(* IEC 61131-3 sources: moqui-plc/simatic-ax/src/moqui/runtime/component/mantle-hvac/src/main/mantle/hvac, 4 files *)

(* ---- MainStatus.st ---- *)
TYPE MainStatus : (
	Standby,
    Ventilation,
    Cooling,
    Heating,
	Drying,
    Fault
); END_TYPE

(* ---- Main.st ---- *)
(*
 * NOTE: In general, the Main component implements the control logic of automated industrial systems (Finite State Machine - FSM)
 * using hierarchical control architectures. It separates control policies from implementation mechanisms,
 * and diagnostic mechanisms from failure/error reaction and system reset policies.
*)

(* Example of a supervisor FSM for a civil HVAC air-handling unit (AHU).
 *
 * Topology:
 *   Mode A Thermostat cooling -> Cooling
 *   Mode B Cooling with RH% dehumidification -> Cooling  (rhControlEnabled=TRUE)
 *   Mode C Winter heating -> Heating
 *   Mode D Heating with RH% control -> Heating (rhControlEnabled=TRUE)
 *   Mode E Interval dehumidification (on/off) -> Drying
 *   Mode F Dehumidification by RH% target -> Drying (rhControlEnabled=TRUE)
 *
 * Output function - which device groups are enabled per state:
 *
 *   State          Cold Group   Hot Group   AHU Fan   Air Flow
 *   -
 *   Standby            OFF         OFF        OFF       OFF
 *   Ventilation        OFF         OFF        ON        ON
 *   Cooling            ON          OFF        ON        ON
 *   Heating            OFF         ON         ON        ON
 *   Drying             ON          ON         ON        ON
 *   Fault              OFF         OFF        OFF       OFF
 *
 * MainRuleEngine generates transition requests; Main consumes them.
 * DeviceManager orchestrates the individual device FBs.
 *
 * Call order in the PLC task:
 *   InputSignalUpdate -> Main -> DeviceManager -> OutputSignalUpdate
 *)
FUNCTION_BLOCK Main
	VAR_EXTERNAL
		clks : Clocks;
		dev : DeviceFacade;
	END_VAR
	VAR_INPUT
		operationType : OperatingMode;
		enable : BOOL;
		deviceConfigContextResetRequest : BOOL := FALSE;
	END_VAR
	VAR_OUTPUT
		done : BOOL;
		error : BOOL;
	END_VAR
	VAR CONSTANT
		componentName : STRING := 'hvac';
	END_VAR
	VAR
		(* Logger facade *)
		logger : LoggerFacade;
		(* FSM transition logic *)
		ruleEngine : MainRuleEngine;
		(* Define a nested FSMs for managing air distribution subsystem. *)
		airDistribCtrl : AirDistributionController;
		(* HAL manager *)
		deviceManager : DeviceManager;
	END_VAR

	(* Logger facade init *)
	logger.enable := TRUE; logger.loggerName := componentName;

	IF NOT enable THEN RETURN; END_IF;

	(* Init: device setup and configuration *)
	IF (operationType = OperatingMode#Init) THEN
		logger(message := 'Setup and configuration of all devices.', level := LogLevel#DEBUG);
		(*
	     * The static device configuration parameters are mapped directly by the device config manager (recipe manager),
		 * while only the dynamic parameters are mapped below in the standby status.
		 *)
		(* Reset signal manager *)
		dev.signalMgmt(operationType := SignalMgmtOperatingMode#Reset, loggerName := componentName);
		dev.status := MainStatus#Standby;
		dev.actualRuntime := UDINT#0;
		dev.actualBreakDuration := UDINT#0;
		dev.processActualDuration := UDINT#0;
		dev.processRemainingDuration := UDINT#0;
		dev.timeBreakEnabled := FALSE;
		dev.isCompleted := FALSE;
		airDistribCtrl(operationType := OperatingMode#Init, enable := FALSE, clock1s := FALSE);
		done := FALSE;
	ELSIF deviceConfigContextResetRequest THEN
		logger(message := 'Reset HVAC device config context.', level := LogLevel#DEBUG);
		(*
	     * Lightweight reset between recipes: keep device init/homing in the Init path,
		 * but clear runtime state inherited from the previous device config.
	     *)
		dev.status := MainStatus#Standby;
		dev.lastStatus := MainStatus#Standby;
		dev.actualRuntime := UDINT#0;
		dev.actualBreakDuration := UDINT#0;
		dev.processActualDuration := UDINT#0;
		dev.processRemainingDuration := UDINT#0;
		dev.timeBreakEnabled := FALSE;
		dev.isCompleted := FALSE;
		airDistribCtrl(operationType := OperatingMode#Init, enable := FALSE, clock1s := FALSE);
		done := FALSE;
	ELSE
		(* FSM transition-condition rule engine *)
		logger(message := 'Run FSM transition-condition logic.', level := LogLevel#DEBUG);
		ruleEngine(operationType := operationType);
	END_IF;

		(*
		 * Preserve the originating phase while idling in Standby so thermostat-driven
		 * Heating/Cooling recipes can stop/start repeatedly until isCompleted becomes TRUE.
		 * Init still stamps Standby, which keeps fresh-start logic for a newly loaded recipe.
	     *)
		IF (operationType = OperatingMode#Init) OR (dev.status <> MainStatus#Standby) THEN
			dev.lastStatus := dev.status;
		END_IF;

	(* Fault overrides any other state *)
	IF dev.faultRequest THEN dev.status := MainStatus#Fault; END_IF;

	(* Main FSM - Output function + State-update function *)
	logger(message := 'Run Main FSM.', level := LogLevel#DEBUG);
	CASE dev.status OF
	    (* Standby / Homing: all groups off, wait for the next phase request. *)
		MainStatus#Standby :
			logger(message := 'Standby.', level := LogLevel#DEBUG);
			dev.standbyRequest := FALSE;

			(* FSM Output function - everything disabled *)
			dev.coldGroupEnableRequest := FALSE;
			dev.coldGroupDisableRequest := TRUE;
			dev.hotGroupEnableRequest := FALSE;
			dev.hotGroupDisableRequest := TRUE;
			dev.ahuFanEnableRequest := FALSE;
			dev.airFlowEnableRequest := FALSE;
			dev.airFlowDisableRequest := TRUE;

			(* FSM status update function *)
			IF dev.ventilationRequest THEN
				dev.status := MainStatus#Ventilation;
			ELSIF dev.coolingRequest THEN
				dev.status := MainStatus#Cooling;
			ELSIF dev.heatingRequest THEN
				dev.status := MainStatus#Heating;
			ELSIF dev.dryingRequest THEN
				dev.status := MainStatus#Drying;
			END_IF;

	    (* Ventilation: AHU + air flow control only - no temperature conditioning. *)
		MainStatus#Ventilation :
			logger(message := 'Ventilation.', level := LogLevel#DEBUG);
			dev.ventilationRequest := FALSE;

			(* FSM output function *)
			dev.coldGroupEnableRequest := FALSE;
			dev.coldGroupDisableRequest := TRUE;
			dev.hotGroupEnableRequest := FALSE;
			dev.hotGroupDisableRequest := TRUE;
			dev.ahuFanEnableRequest := TRUE;
			dev.airFlowEnableRequest := TRUE;
			dev.airFlowDisableRequest := FALSE;

			(* FSM status update function *)
			IF dev.standbyRequest THEN
				dev.status := MainStatus#Standby;
			ELSIF dev.coolingRequest THEN
				dev.status := MainStatus#Cooling;
			ELSIF dev.heatingRequest THEN
				dev.status := MainStatus#Heating;
			ELSIF dev.dryingRequest THEN
				dev.status := MainStatus#Drying;
			END_IF;

	    (*
	     * Cooling: cold group + AHU + air flow control.
	     * Phase 0 (no RH ctrl) and Phase 1 (with RH ctrl, rhControlEnabled=TRUE).
	     * In Phase 1 the hot group is also enabled to post-heat after dehumidification;
	     * that secondary enable is issued by MainRuleEngine via heatingRequest/dryingRequest
	     * transitions rather than here, keeping output function clean.
	     *)
		MainStatus#Cooling :
			logger(message := 'Cooling.', level := LogLevel#DEBUG);
			dev.coolingRequest := FALSE;

			(* FSM output function *)
			dev.coldGroupEnableRequest := TRUE;
			dev.coldGroupDisableRequest := FALSE;
			dev.hotGroupEnableRequest := FALSE;
			dev.hotGroupDisableRequest := TRUE;
			dev.ahuFanEnableRequest := TRUE;
			dev.airFlowEnableRequest := TRUE;
			dev.airFlowDisableRequest := FALSE;

			(* FSM status update function *)
			IF dev.standbyRequest THEN
				dev.status := MainStatus#Standby;
			ELSIF dev.dryingRequest THEN
				dev.status := MainStatus#Drying;
			ELSIF dev.ventilationRequest THEN
				dev.status := MainStatus#Ventilation;
			END_IF;

	    (*
	     * Heating: hot group + AHU + air flow control.
	     * Phase 2 (no RH ctrl) and Phase 3 (with RH ctrl).
	     *)
		MainStatus#Heating :
			logger(message := 'Heating.', level := LogLevel#DEBUG);
			dev.heatingRequest := FALSE;

			(* FSM output function *)
			dev.coldGroupEnableRequest := FALSE;
			dev.coldGroupDisableRequest := TRUE;
			dev.hotGroupEnableRequest := TRUE;
			dev.hotGroupDisableRequest := FALSE;
			dev.ahuFanEnableRequest := TRUE;
			dev.airFlowEnableRequest := TRUE;
			dev.airFlowDisableRequest := FALSE;

			(* FSM status update function *)
			IF dev.standbyRequest THEN
				dev.status := MainStatus#Standby;
			ELSIF dev.dryingRequest THEN
				dev.status := MainStatus#Drying;
			ELSIF dev.ventilationRequest THEN
				dev.status := MainStatus#Ventilation;
			END_IF;

	    (*
	     * Drying: cold + hot + AHU + air flow control.
	     * Phase 4 (time-based run/break) and Phase 5 (RH% controlled).
	     * During break the rule engine transitions to Standby; returns here
	     * when the break is complete.
	     *)
		MainStatus#Drying :
			logger(message := 'Drying.', level := LogLevel#DEBUG);
			dev.dryingRequest := FALSE;

			(* FSM output function *)
			dev.coldGroupEnableRequest := TRUE;
			dev.coldGroupDisableRequest := FALSE;
			dev.hotGroupEnableRequest := TRUE;
			dev.hotGroupDisableRequest := FALSE;
			dev.ahuFanEnableRequest := TRUE;
			dev.airFlowEnableRequest := TRUE;
			dev.airFlowDisableRequest := FALSE;

			(* FSM status update function *)
			IF dev.standbyRequest THEN
				dev.status := MainStatus#Standby;
			ELSIF dev.heatingRequest THEN
				dev.status := MainStatus#Heating;
			ELSIF dev.coolingRequest THEN
				dev.status := MainStatus#Cooling;
			ELSIF dev.ventilationRequest THEN
				dev.status := MainStatus#Ventilation;
			END_IF;

	    (* Fault: all groups off; wait for signal manager to clear all alarms. *)
		MainStatus#Fault :
			logger(message := 'Fault.', level := LogLevel#DEBUG);
			dev.faultRequest := FALSE;

			(* FSM output function *)
			error := TRUE;
			dev.coldGroupEnableRequest := FALSE;
			dev.coldGroupDisableRequest := TRUE;
			dev.hotGroupEnableRequest := FALSE;
			dev.hotGroupDisableRequest := TRUE;
			dev.ahuFanEnableRequest := FALSE;
			dev.airFlowEnableRequest := FALSE;
			dev.airFlowDisableRequest := TRUE;

			(* Return to Standby only when all alarms have been cleared *)
			IF (dev.signalMgmt.cumulativeOutputAction = DWORD#16#0000) THEN
				error := FALSE;
				dev.status := MainStatus#Standby;
			END_IF;
	END_CASE;

	(*
	 * Air distribution is a subordinate subsystem:
	 * it runs only when the main FSM requests air flow and the recipe explicitly
	 * enables alternating high/low air distribution.
	 *)
	airDistribCtrl(
		operationType := operationType,
		enable := dev.airFlowEnableRequest AND dev.airDistributionEnabled,
		clock1s := clks.clock1s);

	done := dev.isCompleted;

	(* Device orchestration (HAL) *)
	logger(message := 'Update HVAC devices.', level := LogLevel#DEBUG);
	deviceManager(operationType := operationType);
	END_FUNCTION_BLOCK

(* ---- MainRuleEngine.st ---- *)
(*
 * MainRuleEngine - transition-condition logic for the HVAC supervisor FSM.
 *
 * Responsibilities:
 *   1. Reset transition requests to safe defaults.
 *   2. Run the signal management engine (fault / alarm / warning detection).
 *   3. Compute boolean predicates from sensor feedback and recipe setpoints.
 *   4. Implement the per-state transition-condition rules.
 *
 * Default / persistence convention
 * At the top of every scan standbyRequest is set TRUE (safe default).
 * Each ACTIVE-state CASE block MUST:
 *   • Set standbyRequest := FALSE (keep current state) in the ELSE branch.
 *   • Set standbyRequest := TRUE (or leave as-is) when an EXIT condition is met.
 *   • Set standbyRequest := FALSE and another*Request := TRUE to switch phase.
 *
 * Without the ELSE branch the system would exit any active state to Standby
 * on the very first scan - a single-scan flash rather than a persistent phase.
 *
 * Process phases:
 *   Phase 0 Thermostat Cooling -> Cooling
 *   Phase 1 Cooling with RH% control -> Cooling (rhControlEnabled)
 *   Phase 2 Heating without RH% control -> Heating
 *   Phase 3 Heating with RH% control -> Heating (rhControlEnabled)
 *   Phase 4 Timed Drying (on/off) -> Drying <-> Standby (break)
 *   Phase 5 Drying with RH% control -> Drying (rhControlEnabled)
 *
 * Duct safety (duct sensors):
 *   The duct T+RH sensor monitors supply-air conditions before the air
 *   enters the curing room. Limit violations raise alarms to protect
 *   product (≈ €80-90 k of salami/prosciutto on trolleys).
 *   ductTempOverMax -> air too hot -> ImmediateStop (protects product)
 *   ductTempUnderMin -> air too cold -> ImmediateStop (protects product)
 *   ductRhOverMax -> saturated -> Warning only (condensation risk)
 *)
FUNCTION_BLOCK MainRuleEngine
	VAR_EXTERNAL
		clks : Clocks;
		dev : DeviceFacade;
	END_VAR
	VAR_INPUT
		operationType : OperatingMode := OperatingMode#Run;
	END_VAR
	VAR_OUTPUT
		error : BOOL;
	END_VAR
	VAR
		(* Device diagnostics *)
		deviceDiags : DeviceDiagnostics;
		tempDeviation : REAL;
		rhDeviation : REAL;
	END_VAR

	(* Reset transition requests to safe defaults.
	 *
	 * standbyRequest = TRUE  -> return to / stay in Standby (safe default).
	 * Active-state CASE blocks override to FALSE to keep the current phase alive,
	 * or set another *Request to switch phases.
	 *)
	dev.faultRequest := FALSE;
	dev.standbyRequest := TRUE;
	dev.heatingRequest := FALSE;
	dev.coolingRequest := FALSE;
	dev.ventilationRequest := FALSE;
	dev.dryingRequest := FALSE;

	deviceDiags(operationType := operationType, error => error);

	(* Compute sensor predicates *)

	(* Process temperature sensor *)
	dev.tempInRange := (dev.tempFeedback >= dev.tempMin + dev.tempHysteresis)
		AND (dev.tempFeedback <= dev.tempMax - dev.tempHysteresis);
	tempDeviation := dev.tempFeedback - dev.tempSetpoint;
	IF tempDeviation < REAL#0.0 THEN
		tempDeviation := -tempDeviation;
	END_IF;
	dev.tempAtSetpoint := tempDeviation <= dev.tempHysteresis;
	dev.tempOverMax := dev.tempFeedback > dev.tempMax;
	dev.tempOverMin := dev.tempFeedback > dev.tempMin;
	dev.tempUnderMin := dev.tempFeedback < dev.tempMin;
	dev.tempUnderMax := dev.tempFeedback < dev.tempMax;
	(* Process RH sensor *)
	rhDeviation := dev.rhFeedback - dev.rhSetpoint;
	IF rhDeviation < REAL#0.0 THEN
		rhDeviation := -rhDeviation;
	END_IF;
	dev.rhAtSetpoint := rhDeviation <= dev.rhHysteresis;
	dev.rhOverMax := dev.rhFeedback > dev.rhMax - dev.rhHysteresis;
	dev.rhUnderMin := dev.rhFeedback < dev.rhMin + dev.rhHysteresis;
	dev.rhOverMin := dev.rhFeedback > dev.rhMin;
	dev.rhUnderMax := dev.rhFeedback < dev.rhMax;

	(* Duct sensor - safety predicates *)
	dev.ductTempOverMax := dev.ductTempFeedback > dev.ductTempMax;
	dev.ductTempUnderMin := dev.ductTempFeedback < dev.ductTempMin;
	dev.ductRhOverMax := dev.ductRhFeedback > dev.ductRhMax;

	(*
	 * Process timing - run / break cycle.
	 *
	 * processActualDuration must NOT advance while the FSM is in Standby
	 * waiting for a phase to start (i.e. not in a break).
	 * If it did, isCompleted could fire while the process has not yet begun,
	 * causing the phase to complete immediately without doing any work.
	 *
	 * Counting rules:
	 *   Break  (timeBreakEnabled=TRUE, status=Standby): advance processActualDuration + actualBreakDuration.
	 *   Active (status ≠ Standby):                      advance processActualDuration + actualRuntime.
	 *   Idle   (status=Standby, NOT timeBreakEnabled):  no counters advance.
	 *)
	IF clks.clock1s THEN
		IF dev.timeBreakEnabled AND dev.status = MainStatus#Standby THEN
			(* Break counting *)
			dev.processActualDuration := dev.processActualDuration + UDINT#1;
			dev.actualBreakDuration := dev.actualBreakDuration + UDINT#1;
			IF dev.estimatedBreakDuration > UDINT#0 THEN
				(* Break ends when both minimum and estimated durations are met; reset counters for next run *)
				IF (dev.actualBreakDuration >= dev.estimatedBreakDuration)
						AND (dev.actualBreakDuration >= dev.minBreakDuration) THEN
					dev.timeBreakEnabled := FALSE;
					dev.actualRuntime := UDINT#0;
					dev.actualBreakDuration := UDINT#0;
				END_IF;
			END_IF;
		ELSIF dev.status <> MainStatus#Standby THEN
			(* Active run counting - only while the FSM is in an active phase state *)
			dev.processActualDuration := dev.processActualDuration + UDINT#1;
			dev.actualRuntime := dev.actualRuntime + UDINT#1;
			IF dev.estimatedRuntime > UDINT#0 THEN
				dev.processRemainingDuration := dev.processEstimatedDuration - dev.processActualDuration;
				IF NOT dev.timeBreakEnabled
						AND (dev.actualRuntime >= dev.estimatedRuntime)
						AND (dev.actualRuntime >= dev.minRuntime) THEN
					dev.timeBreakEnabled := TRUE;
					dev.actualBreakDuration := UDINT#0;
				END_IF;
			END_IF;
		ELSIF (dev.lastStatus = MainStatus#Cooling OR dev.lastStatus = MainStatus#Heating)
				AND NOT dev.isCompleted THEN
			(* Thermostat dwell between active cycles counts toward phase duration,
			 * but does not count as active runtime. *)
			dev.processActualDuration := dev.processActualDuration + UDINT#1;
			IF dev.processEstimatedDuration > UDINT#0 THEN
				dev.processRemainingDuration := dev.processEstimatedDuration - dev.processActualDuration;
			END_IF;
		END_IF;

		(* isCompleted is independent of the run/break cycle:
		 * a phase with only processEstimatedDuration set (no run/break) must also complete. *)
		IF dev.processEstimatedDuration > UDINT#0 THEN
			dev.isCompleted :=
				(dev.processActualDuration >= dev.processEstimatedDuration)
				AND (dev.processActualDuration >= dev.processMinDuration);
		END_IF;
	END_IF;

	(* Fault gate *)
	IF error OR ((dev.signalMgmt.cumulativeOutputAction AND DWORD#16#0002) <> DWORD#16#0000) THEN
		dev.faultRequest := TRUE;
		RETURN;
	END_IF;

	(*
	 * Transition-condition rule engine
	 *
	 * Persistence rule: every active-state CASE MUST end with
	 *   ELSE dev.standbyRequest := FALSE; [ keep current state alive ]
	 * to prevent the scan-level default (standbyRequest=TRUE) from immediately
	 * bouncing the FSM back to Standby before the exit condition is reached.
	 *)
	CASE dev.status OF
	    (*
	     * Standby - decide next phase.
	     * Default standbyRequest=TRUE keeps the system here.
	     * Override when an external condition requires re-entering a phase.
	     *)
		MainStatus#Standby :
			(*
			 * Transition-condition evaluation order:
			 *   1. Safety overrides (cooling/heating if temperature out of limits).
			 *   2. Phase-resume conditions (drying after break, thawing).
			 *   3. Fresh-start drying (new recipe loaded, lastStatus=Standby after Init).
			 *   4. Hold-in-Standby (isCompleted or core setpoint reached) — checked LAST.
			 *
			 * isCompleted is evaluated last so that phase-transition conditions are always
			 * reachable.  The guard dev.lastStatus=Standby in condition 3 makes it safe:
			 * that guard is only TRUE after Init has run (Init sets dev.status=Standby, so
			 * line-97 lastStatus:=status writes Standby), which also resets isCompleted=FALSE.
			 * In the one-scan gap between a phase exit (isCompleted=TRUE, lastStatus=Cooling/
			 * Drying/…) and Init, lastStatus≠Standby, so condition 3 cannot fire, and
			 * condition 4 correctly holds the FSM in Standby until configMgmt advances.
			 *)
			IF (dev.lastStatus = MainStatus#Cooling OR dev.lastStatus = MainStatus#Standby)
					AND dev.tempOverMax THEN
				(* Temperature above limit -> start/resume cooling *)
				dev.standbyRequest := FALSE;
				dev.coolingRequest := TRUE;

			ELSIF (dev.lastStatus = MainStatus#Heating OR dev.lastStatus = MainStatus#Standby)
					AND dev.tempUnderMin THEN
				(* Temperature below limit -> start/resume heating *)
				dev.standbyRequest := FALSE;
				dev.heatingRequest := TRUE;

			ELSIF dev.lastStatus = MainStatus#Drying
					AND NOT dev.timeBreakEnabled
					AND NOT dev.isCompleted
					AND dev.tempInRange
					AND (NOT dev.rhControlOnly
					OR (dev.rhControlEnabled AND dev.rhOverMax)) THEN
				(*
				 * End of break: resume drying run when all conditions are met:
				 *   - break elapsed (NOT timeBreakEnabled)
				 *   - process not yet complete (NOT isCompleted)
				 *   - temperature back in process window (tempInRange)
				 *   - humidity still needs treatment
				 *)
				dev.standbyRequest := FALSE;
				dev.dryingRequest := TRUE;

			ELSIF dev.lastStatus = MainStatus#Standby
					AND NOT dev.tempOverMax
					AND dev.rhOverMax THEN
				(*
				 * Fresh drying recipe loaded: start drying when temperature is safe (≤ tempMax)
				 * and humidity needs treatment.
				 *
				 * NOT tempOverMax (instead of tempInRange) eliminates the dead zone at
				 * tempFeedback ∈ (tempMax-hyst, tempMax] that would leave the FSM stuck in
				 * Standby after a cooling phase delivered temp near the top of the window.
				 * If temp is below tempMin the Drying state switches to Heating temporarily,
				 * then returns to Drying once tempOverMin.
				 *)
				dev.standbyRequest := FALSE;
				dev.dryingRequest := TRUE;

			ELSIF dev.isCompleted THEN
				dev.standbyRequest := TRUE; (* Explicit: work done, hold here until configMgmt advances *)

			(* No ELSE needed here: standbyRequest=TRUE default holds Standby *)
			END_IF;

	    (*
	     * Ventilation - AHU + air flow only.
	     * No automatic exit; operator or recipe change triggers Standby.
	     *)
		MainStatus#Ventilation :
			IF dev.isCompleted THEN
				dev.standbyRequest := TRUE;
			ELSE
				dev.standbyRequest := FALSE; (* Keep ventilating *)
			END_IF;

	    (*
	     * Cooling - cold group + AHU.
	     * Phase 0: thermostat-only (no RH control).
	     * Phase 1: with RH control - when RH reaches setpoint switch to Drying.
	     *
	     * EXIT conditions (standbyRequest=TRUE):
	     *   tempUnderMin -> target reached, stop cooling.
	     *   isCompleted -> work-effort complete.
	     * SWITCH conditions (standbyRequest=FALSE):
	     *   lastStatus=Drying + tempUnderMax -> resume drying.
	     *   lastStatus=Drying + tempUnderMax -> resume drying.
	     * ELSE -> keep cooling (temperature still above tempMin).
	     *)
		MainStatus#Cooling :
			IF dev.tempUnderMin OR dev.isCompleted THEN
				dev.standbyRequest := TRUE;
			ELSIF dev.lastStatus = MainStatus#Drying
					AND (dev.tempUnderMax
					OR (dev.rhControlEnabled AND dev.rhOverMax AND dev.tempUnderMax)) THEN
				dev.standbyRequest := FALSE;
				dev.dryingRequest := TRUE;
			ELSE
				dev.standbyRequest := FALSE; (* Keep cooling - tempFeedback still above tempMin *)
			END_IF;

	    (*
	     * Heating - hot group + AHU.
	     * Phase 2 (no RH ctrl) / Phase 3 (with RH ctrl).
	     *
	     * EXIT: tempOverMax, isCompleted, or core temperature reached.
	     * SWITCH to Drying: temperature restored to process window.
	     * ELSE: keep heating.
	     *)
		MainStatus#Heating :
			IF dev.isCompleted OR dev.tempOverMax THEN
				dev.standbyRequest := TRUE;
			ELSIF (dev.lastStatus = MainStatus#Drying AND dev.tempOverMin)
					OR (dev.rhControlEnabled AND dev.rhOverMax) THEN
				dev.standbyRequest := FALSE;
				dev.dryingRequest  := TRUE;
			ELSE
				dev.standbyRequest := FALSE; (* Keep heating - tempFeedback still below tempMax *)
			END_IF;

	    (*
	     * Drying - cold + hot + AHU (Phase 4 / Phase 5).
	     *
	     * Normal end conditions:
	     *   Time-based (!rhControlOnly): T in range AND runtime elapsed.
	     *   RH-only: RH ≤ rhMin AND minimum runtime elapsed.
	     *   RH+time: RH ≤ rhMin (timer managed externally).
	     *   isCompleted: work-effort done.
	     * Break trigger: timeBreakEnabled -> Standby (returns here after break).
	     * Override to Cooling: tempOverMax.
	     * Override to Heating: tempUnderMin.
	     * ELSE: keep drying.
	     *)
		MainStatus#Drying :
			IF dev.isCompleted THEN
				dev.standbyRequest := TRUE;
			ELSIF NOT dev.rhControlOnly
					AND dev.tempInRange
					AND (dev.estimatedRuntime > UDINT#0)
					AND (dev.actualRuntime > dev.estimatedRuntime) THEN
				dev.standbyRequest := TRUE; (* Time-based running completed *)
			ELSIF dev.rhControlOnly
					AND dev.rhUnderMin
					AND (dev.actualRuntime >= dev.minRuntime) THEN
				dev.standbyRequest := TRUE; (* RH-only target reached *)
			ELSIF dev.rhControlEnabled AND dev.rhUnderMin THEN
				dev.standbyRequest := TRUE; (* RH+time: humidity at minimum *)
			ELSIF dev.timeBreakEnabled THEN
				dev.standbyRequest := TRUE; (* Begin break - rule engine resumes Drying after break *)
			ELSIF dev.tempOverMax THEN
				dev.standbyRequest := FALSE;
				dev.coolingRequest := TRUE;  (* Temporary cooling override *)
			ELSIF dev.tempUnderMin THEN
				dev.standbyRequest := FALSE;
				dev.heatingRequest := TRUE;  (* Temporary heating override *)
			ELSE
				dev.standbyRequest := FALSE; (* Keep drying - process ongoing *)
			END_IF;

	END_CASE;
	END_FUNCTION_BLOCK

(* ---- ParameterLogger.st ---- *)
(*
 * Periodic logger for the numeric parameters of the HVAC Application.
 *
 * Physical signal logging belongs to InputSignalUpdate and OutputSignalUpdate.
 * This block logs the logical values exposed through DeviceFacade. The source
 * of each event is the exact moqui.math.Parameter.parameterId from
	 * HVACDemoData.xml; loggerName is the owning Device.deviceId.
 *)
FUNCTION_BLOCK ParameterLogger
	VAR_EXTERNAL
		dev : DeviceFacade;
		clks : Clocks;
	END_VAR
	VAR_INPUT
		operationType : OperatingMode;
	END_VAR
	VAR
		logger : LoggerFacade;
	END_VAR
	VAR CONSTANT
		componentName : STRING := 'HVAC_DEMO_PLC';
	END_VAR

	(* Log only one snapshot per minute, independently of the PLC task cycle. *)
	IF (operationType <> OperatingMode#Run) OR NOT clks.clock1minute THEN RETURN; END_IF;

	logger.enable := TRUE;
	logger.loggerName := componentName;
	logger.payloadType := LogPayloadType#Numeric;
	logger.level := LogLevel#Info;

	(* Process setpoints and limits. *)
	logger(source := 'HvacTempSetpoint', numericValue := TO_LREAL(dev.tempSetpoint));
	logger(source := 'HvacTempHysteresis', numericValue := TO_LREAL(dev.tempHysteresis));
	logger(source := 'HvacTempMin', numericValue := TO_LREAL(dev.tempMin));
	logger(source := 'HvacTempMax', numericValue := TO_LREAL(dev.tempMax));
	logger(source := 'HvacRhSetpoint', numericValue := TO_LREAL(dev.rhSetpoint));
	logger(source := 'HvacRhHysteresis', numericValue := TO_LREAL(dev.rhHysteresis));
	logger(source := 'HvacRhMin', numericValue := TO_LREAL(dev.rhMin));
	logger(source := 'HvacRhMax', numericValue := TO_LREAL(dev.rhMax));
	logger(source := 'HvacDuctTempMin', numericValue := TO_LREAL(dev.ductTempMin));
	logger(source := 'HvacDuctTempMax', numericValue := TO_LREAL(dev.ductTempMax));
	logger(source := 'HvacDuctRhMax', numericValue := TO_LREAL(dev.ductRhMax));
	(* Application timing parameters and runtime counters. *)
	logger(source := 'HvacSetPointTimeHigh', numericValue := TO_LREAL(dev.setPointTimeHigh));
	logger(source := 'HvacSetPointTimeLow', numericValue := TO_LREAL(dev.setPointTimeLow));
	logger(source := 'HvacEstimatedRuntime', numericValue := TO_LREAL(dev.estimatedRuntime));
	logger(source := 'HvacMinRuntime', numericValue := TO_LREAL(dev.minRuntime));
	logger(source := 'HvacEstimatedBreakDuration', numericValue := TO_LREAL(dev.estimatedBreakDuration));
	logger(source := 'HvacMinBreakDuration', numericValue := TO_LREAL(dev.minBreakDuration));
	logger(source := 'HvacProcessEstimatedDuration', numericValue := TO_LREAL(dev.processEstimatedDuration));
	logger(source := 'HvacProcessMinDuration', numericValue := TO_LREAL(dev.processMinDuration));
	logger(source := 'HvacProcessRemainingDuration', numericValue := TO_LREAL(dev.processRemainingDuration));
	logger(source := 'HvacProcessActualDuration', numericValue := TO_LREAL(dev.processActualDuration));
	logger(source := 'HvacActualRuntime', numericValue := TO_LREAL(dev.actualRuntime));
	logger(source := 'HvacActualBreakDuration', numericValue := TO_LREAL(dev.actualBreakDuration));
	(* Numeric machine references. *)
	logger(source := 'HvacAhuFanSpeedSetpoint', numericValue := TO_LREAL(dev.ahuFanSpeedSetpoint));
	logger(source := 'HvacAirFlowRef', numericValue := TO_LREAL(dev.airFlowRef));
	(* Process measurements. *)
	logger(source := 'HvacTempFeedback', numericValue := TO_LREAL(dev.tempFeedback));
	logger(source := 'HvacRhFeedback', numericValue := TO_LREAL(dev.rhFeedback));
	logger(source := 'HvacDuctTempFeedback', numericValue := TO_LREAL(dev.ductTempFeedback));
	logger(source := 'HvacDuctRhFeedback', numericValue := TO_LREAL(dev.ductRhFeedback));
END_FUNCTION_BLOCK
